PROGRAM faults
VAR PERSISTENT

//---Equipment Failure Faults----------------------------------------------------------------------------------------------

	//Discrete alarm example.  Replace with your own alarms
	u_3112_fail_to_start : alarm;
	u_3212_fail_to_start : alarm;
	u_3312_fail_to_start : alarm;
	u_3160_fail_to_start : alarm;
	u_3260_fail_to_start : alarm;
	u_3360_fail_to_start : alarm;
	u_3370_fail_to_start : alarm;
	u_3405_fail_to_start : alarm;
	// Discrete Alarm Example
	u_3112_fail_to_stop: Alarm;
	u_3212_fail_to_stop: Alarm;
	u_3312_fail_to_stop: Alarm;
	u_3160_fail_to_stop: Alarm;
	u_3260_fail_to_stop: Alarm;
	u_3360_fail_to_stop: Alarm;
	u_3370_fail_to_stop: Alarm;
	u_3405_fail_to_stop: Alarm;

	// Example analog valve position fail alarm
	av_3148_position_fail: Alarm;
	// Example digital valve fail to open alarm
	nv_3372_fail_to_open: Alarm;
	// Example digital valve fail to close alarm
	nv_3372_fail_to_close: Alarm;
	
//---System threshold alarms------------------------------------------------------------------------------------------------

	// Analog alarm low low
	cct_3120_low_low: Alarm;
	cct_3142_low_low: Alarm;
	cct_3220_low_low: Alarm;
	cct_3242_low_low: Alarm;
	cct_3320_low_low: Alarm;
	cct_3342_low_low: Alarm;
	cct_3413_low_low: Alarm;
	cgt_3910_low_low: Alarm;
	cpt_3144_low_low: Alarm;
	cpt_3158_low_low: Alarm;
	cpt_3407_low_low: Alarm;
	et_3711_low_low: Alarm;
	ft_3122_low_low: Alarm;
	ft_3222_low_low: Alarm;
	ft_3322_low_low: Alarm;
	it_3702_low_low: Alarm;
	lit_3905_low_low: Alarm;
	lit_3906_low_low: Alarm;
	lit_3907_low_low: Alarm;
	lit_3908_low_low: Alarm;
	lit_3915_low_low: Alarm;
	lt_3102_low_low: Alarm;
	lt_3153_low_low: Alarm;
	lt_3202_low_low: Alarm;
	lt_3253_low_low: Alarm;
	lt_3302_low_low: Alarm;
	lt_3353_low_low: Alarm;
	lt_3402_low_low: Alarm;
	pt_3119_low_low: Alarm;
	pt_3141_low_low: Alarm;
	pt_3219_low_low: Alarm;
	pt_3241_low_low: Alarm;
	pt_3319_low_low: Alarm;
	pt_3341_low_low: Alarm;
	pt_3414_low_low: Alarm;
	pt_3428_low_low: Alarm;
	tt_3118_low_low: Alarm;
	tt_3140_low_low: Alarm;
	tt_3218_low_low: Alarm;
	tt_3240_low_low: Alarm;
	tt_3318_low_low: Alarm;
	tt_3340_low_low: Alarm;
	tt_3432_low_low: Alarm;
	tt_3601_low_low: Alarm;


	// Analog alarm low
	cct_3120_low: Alarm;
	cct_3142_low: Alarm;
	cct_3220_low: Alarm;
	cct_3242_low: Alarm;
	cct_3320_low: Alarm;
	cct_3342_low: Alarm;
	cct_3413_low: Alarm;
	cgt_3910_low: Alarm;
	cpt_3144_low: Alarm;
	cpt_3158_low: Alarm;
	cpt_3407_low: Alarm;
	et_3711_low: Alarm;
	ft_3122_low: Alarm;
	ft_3222_low: Alarm;
	ft_3322_low: Alarm;
	it_3702_low: Alarm;
	lit_3905_low: Alarm;
	lit_3906_low: Alarm;
	lit_3907_low: Alarm;
	lit_3908_low: Alarm;
	lit_3915_low: Alarm;
	lt_3102_low: Alarm;
	lt_3153_low: Alarm;
	lt_3202_low: Alarm;
	lt_3253_low: Alarm;
	lt_3302_low: Alarm;
	lt_3353_low: Alarm;
	lt_3402_low: Alarm;
	pt_3119_low: Alarm;
	pt_3141_low: Alarm;
	pt_3219_low: Alarm;
	pt_3241_low: Alarm;
	pt_3319_low: Alarm;
	pt_3341_low: Alarm;
	pt_3414_low: Alarm;
	pt_3428_low: Alarm;
	tt_3118_low: Alarm;
	tt_3140_low: Alarm;
	tt_3218_low: Alarm;
	tt_3240_low: Alarm;
	tt_3318_low: Alarm;
	tt_3340_low: Alarm;
	tt_3432_low: Alarm;
	tt_3601_low: Alarm;


	// Analog alarm high
		cct_3120_high: Alarm;
	cct_3142_high: Alarm;
	cct_3220_high: Alarm;
	cct_3242_high: Alarm;
	cct_3320_high: Alarm;
	cct_3342_high: Alarm;
	cct_3413_high: Alarm;
	cgt_3910_high: Alarm;
	cpt_3144_high: Alarm;
	cpt_3158_high: Alarm;
	cpt_3407_high: Alarm;
	et_3711_high: Alarm;
	ft_3122_high: Alarm;
	ft_3222_high: Alarm;
	ft_3322_high: Alarm;
	it_3702_high: Alarm;
	lit_3905_high: Alarm;
	lit_3906_high: Alarm;
	lit_3907_high: Alarm;
	lit_3908_high: Alarm;
	lit_3915_high: Alarm;
	lt_3102_high: Alarm;
	lt_3153_high: Alarm;
	lt_3202_high: Alarm;
	lt_3253_high: Alarm;
	lt_3302_high: Alarm;
	lt_3353_high: Alarm;
	lt_3402_high: Alarm;
	pt_3119_high: Alarm;
	pt_3141_high: Alarm;
	pt_3219_high: Alarm;
	pt_3241_high: Alarm;
	pt_3319_high: Alarm;
	pt_3341_high: Alarm;
	pt_3414_high: Alarm;
	pt_3428_high: Alarm;
	tt_3118_high: Alarm;
	tt_3140_high: Alarm;
	tt_3218_high: Alarm;
	tt_3240_high: Alarm;
	tt_3318_high: Alarm;
	tt_3340_high: Alarm;
	tt_3432_high: Alarm;
	tt_3601_high: Alarm;


	// Analog alarm high high
		cct_3120_high_high: Alarm;
	cct_3142_high_high: Alarm;
	cct_3220_high_high: Alarm;
	cct_3242_high_high: Alarm;
	cct_3320_high_high: Alarm;
	cct_3342_high_high: Alarm;
	cct_3413_high_high: Alarm;
	cgt_3910_high_high: Alarm;
	cpt_3144_high_high: Alarm;
	cpt_3158_high_high: Alarm;
	cpt_3407_high_high: Alarm;
	et_3711_high_high: Alarm;
	ft_3122_high_high: Alarm;
	ft_3222_high_high: Alarm;
	ft_3322_high_high: Alarm;
	it_3702_high_high: Alarm;
	lit_3905_high_high: Alarm;
	lit_3906_high_high: Alarm;
	lit_3907_high_high: Alarm;
	lit_3908_high_high: Alarm;
	lit_3915_high_high: Alarm;
	lt_3102_high_high: Alarm;
	lt_3153_high_high: Alarm;
	lt_3202_high_high: Alarm;
	lt_3253_high_high: Alarm;
	lt_3302_high_high: Alarm;
	lt_3353_high_high: Alarm;
	lt_3402_high_high: Alarm;
	pt_3119_high_high: Alarm;
	pt_3141_high_high: Alarm;
	pt_3219_high_high: Alarm;
	pt_3241_high_high: Alarm;
	pt_3319_high_high: Alarm;
	pt_3341_high_high: Alarm;
	pt_3414_high_high: Alarm;
	pt_3428_high_high: Alarm;
	tt_3118_high_high: Alarm;
	tt_3140_high_high: Alarm;
	tt_3218_high_high: Alarm;
	tt_3240_high_high: Alarm;
	tt_3318_high_high: Alarm;
	tt_3340_high_high: Alarm;
	tt_3432_high_high: Alarm;
	tt_3601_high_high: Alarm;



END_VAR

//Instantiate the alarm block, and map the inputs from the OPC GVL
u_3160_fail_to_start();
u_3160_fail_to_start.alm_ack:=opc.popa_0081_alarm_ack;
u_3160_fail_to_start.reset:=opc.popa_0081_alarm_reset;
u_3160_fail_to_start.priority:=opc.popa_0081_u_3160_fail_to_start_priority;
u_3160_fail_to_start.delay_setpoint:=opc.popa_0081_u_3160_fail_to_start_delay_setpoint;
u_3160_fail_to_start.enable:=opc.popa_0081_u_3160_fail_to_start_enable;

//Place your alarm trigger logic here.  
IF motor_starter_control.u_3160.run_command=TRUE AND motor_starter_control.u_3160.run_feedback=FALSE THEN
	u_3160_fail_to_start.trigger:=TRUE;
	ELSE
		u_3160_fail_to_start.trigger:=False;
	END_IF
	
//Instantiate the alarm block, and map the inputs from the OPC GVL
u_3160_fail_to_stop();
u_3160_fail_to_stop.alm_ack:=opc.popa_0081_alarm_ack;
u_3160_fail_to_stop.reset:=opc.popa_0081_alarm_reset;
u_3160_fail_to_stop.priority:=opc.popa_0081_u_3160_fail_to_stop_priority;
u_3160_fail_to_stop.delay_setpoint:=opc.popa_0081_u_3160_fail_to_stop_delay_setpoint;
u_3160_fail_to_stop.enable:=opc.popa_0081_u_3160_fail_to_stop_enable;

//Place your alarm trigger logic here.  
IF motor_starter_control.u_3160.run_command=FALSE AND motor_starter_control.u_3160.run_feedback=TRUE THEN
	u_3160_fail_to_stop.trigger:=TRUE;
	ELSE
		u_3160_fail_to_stop.trigger:=FALSE;
	END_IF
	
//Instantiate the alarm block, and map the inputs from the OPC GVL
u_3112_fail_to_start();
u_3112_fail_to_start.alm_ack:=opc.popa_0081_alarm_ack;
u_3112_fail_to_start.reset:=opc.popa_0081_alarm_reset;
u_3112_fail_to_start.priority:=opc.popa_0081_u_3112_fail_to_start_priority;
u_3112_fail_to_start.delay_setpoint:=opc.popa_0081_u_3112_fail_to_start_delay_setpoint;
u_3112_fail_to_start.enable:=opc.popa_0081_u_3112_fail_to_start_enable;

//Place your alarm trigger logic here.  
IF motor_vfd_control.u_3112.run_command=TRUE AND motor_vfd_control.u_3112.run_feedback=FALSE THEN
	u_3112_fail_to_start.trigger:=TRUE;
	ELSE
		u_3112_fail_to_start.trigger:=FALSE;
	END_IF
	
//Instantiate the alarm block, and map the inputs from the OPC GVL
u_3112_fail_to_stop();
u_3112_fail_to_stop.alm_ack:=opc.popa_0081_alarm_ack;
u_3112_fail_to_stop.reset:=opc.popa_0081_alarm_reset;
u_3112_fail_to_stop.priority:=opc.popa_0081_u_3112_fail_to_stop_priority;
u_3112_fail_to_stop.delay_setpoint:=opc.popa_0081_u_3112_fail_to_stop_delay_setpoint;
u_3112_fail_to_stop.enable:=opc.popa_0081_u_3112_fail_to_stop_enable;

//Place your alarm trigger logic here.  
IF motor_vfd_control.u_3112.run_command=FALSE AND motor_vfd_control.u_3112.run_feedback=TRUE THEN
	u_3112_fail_to_stop.trigger:=TRUE;
	ELSE
		u_3112_fail_to_stop.trigger:=FALSE;
	END_IF
	
//Instantiate the alarm block, and map the inputs from the OPC GVL
av_3148_position_fail();
av_3148_position_fail.alm_ack:=opc.popa_0081_alarm_ack;
av_3148_position_fail.reset:=opc.popa_0081_alarm_reset;
av_3148_position_fail.priority:=opc.popa_0081_av_3148_position_fail_priority;
av_3148_position_fail.delay_setpoint:=opc.popa_0081_av_3148_position_fail_delay_setpoint;
av_3148_position_fail.enable:=opc.popa_0081_av_3148_position_fail_enable;

//Place your alarm trigger logic here.  
IF io_mapping.av_3148_position_feedback.scaled_value>valve_analog_control.av_3148.position_deadband_high OR io_mapping.av_3148_position_feedback.scaled_value<valve_analog_control.av_3148.position_deadband_low THEN
	av_3148_position_fail.trigger:=TRUE;
	ELSE
		av_3148_position_fail.trigger:=FALSE;
	END_IF
	
//Instantiate the alarm block, and map the inputs from the OPC GVL
nv_3372_fail_to_open();
nv_3372_fail_to_open.alm_ack:=opc.popa_0081_alarm_ack;
nv_3372_fail_to_open.reset:=opc.popa_0081_alarm_reset;
nv_3372_fail_to_open.priority:=opc.popa_0081_nv_3372_fail_to_open_priority;
nv_3372_fail_to_open.delay_setpoint:=opc.popa_0081_nv_3372_fail_to_open_delay_setpoint;
nv_3372_fail_to_open.enable:=opc.popa_0081_nv_3372_fail_to_open_enable;

//Place your alarm trigger logic here.  
IF valve_digital_control.nv_3372.open_command=TRUE AND valve_digital_control.nv_3372.open_feedback=FALSE THEN
	nv_3372_fail_to_open.trigger:=TRUE;
	ELSE
		nv_3372_fail_to_open.trigger:=FALSE;
	END_IF
	
//Instantiate the alarm block, and map the inputs from the OPC GVL
nv_3372_fail_to_close();
nv_3372_fail_to_close.alm_ack:=opc.popa_0081_alarm_ack;
nv_3372_fail_to_close.reset:=opc.popa_0081_alarm_reset;
nv_3372_fail_to_close.priority:=opc.popa_0081_nv_3372_fail_to_close_priority;
nv_3372_fail_to_close.delay_setpoint:=opc.popa_0081_nv_3372_fail_to_close_delay_setpoint;
nv_3372_fail_to_close.enable:=opc.popa_0081_nv_3372_fail_to_close_enable;

//Place your alarm trigger logic here.  
IF valve_digital_control.nv_3372.open_command=FALSE AND valve_digital_control.nv_3372.open_feedback=TRUE THEN
	nv_3372_fail_to_close.trigger:=TRUE;
	ELSE
		nv_3372_fail_to_close.trigger:=FALSE;
	END_IF	

	
//---System threshold alarms---------------------------------------------------------------------------------------------------

END_PROGRAM

(* stored: Version 1.1.0.1, ProductVersion 3.1.4024.12
   POU faults: Id {676b0c44-de53-481b-87a6-7f945cc11bcf}, SpecialFunc None *)
